PROGRAM MAIN
VAR
END_VAR

END_PROGRAM

(* stored: Version 1.1.0.1
   POU MAIN: Id {f82431f8-a229-4992-aa97-38fba9da4c4c} *)
